TYPE ST_TX_Python :
STRUCT
	sAuditExportQuery				:STRING[300];
	sAuditFileName					:STRING[300];
	sBatchName						:STRING[300];
END_STRUCT
END_TYPE

(* stored: Version 1.1.0.1, ProductVersion 3.1.4024.12
   DUT ST_TX_Python: Id {5a0841a1-baba-4654-8b4a-1a39f5c7e7d3} *)
